// TIA Portal project "KolosCwiczenieSymulatorow" (V14)

(* hardware
DEVICE "S7-1200 station_1"  S7-1200 Station
   slot 0: "Rack_0"  S7-1200 Rack  Rack  V1.0
   slot 1: "PLC_1"  CPU 1214C DC/DC/DC  6ES7 214-1AG40-0XB0  V4.2
DEVICE "HMI_1"  TP700 Comfort
   slot 0: "TP700 Comfort"  TP700 Comfort  6AV2 124-0GC01-0AX0  14.0.1.0
   slot 1: "HMI_RT_1"  TP700 Comfort  6AV2 124-0GC01-0AX0  14.0.1.0
   slot 5: "HMI_1.IE_CP_1"  PROFINET Interface  14.0.1.0
      slot 1: "PROFINET Interface_1"  PROFINET Interface
         slot 1: "Port_1"  Port
         slot 2: "Port_2"  Port
   slot 7: "HMI_1.MPI/DP_CP_1"  MPI/DP Interface  14.0.1.0
*)

// ===== PLC "PLC_1"  CPU 1214C DC/DC/DC =====

VAR_GLOBAL   // PLC tag table "Default tag table"
   "Otworz zawor" AT %Q0.2 : Bool;
   "Zawor Otwarty" AT %I0.1 : Bool;
   "Zawor zamkniety" AT %I0.2 : Bool;
   "Zamknij zawor" AT %Q0.3 : Bool;
   "Dolej" AT %Q0.4 : Bool;
   "Poziom" AT %IW64 : Word;
   "Clock_Byte" AT %MB0 : Byte;
   "Clock_10Hz" AT %M0.0 : Bool;
   "Clock_5Hz" AT %M0.1 : Bool;
   "Clock_2.5Hz" AT %M0.2 : Bool;
   "Clock_2Hz" AT %M0.3 : Bool;
   "Clock_1.25Hz" AT %M0.4 : Bool;
   "Clock_1Hz" AT %M0.5 : Bool;
   "Clock_0.625Hz" AT %M0.6 : Bool;
   "Clock_0.5Hz" AT %M0.7 : Bool;
   "Wypompuj" AT %Q0.5 : Bool;
   "Tag_1" AT %M10.0 : Bool;
   "Tag_2" AT %M10.1 : Bool;
   "Tag_3" AT %IW68 : Word;
   "Tag_4" AT %I10.0 : Bool;
   "Zawor_otwarty" AT %I10.1 : Bool;
   "Zawor_zamkniety" AT %I10.2 : Bool;
   "Tag_5" AT %IW69 : Word;
   "Tag_6" AT %MD30 : DWord;
   "Moc" AT %QW10 : Word;
   "Tag_8" AT %QD10 : Real;
   "Temperatura" AT %ID30 : Real;
   "Tag_10" AT %M10.3 : Bool;
   "Tag_7" AT %IW30 : Word;
   "Tag_9" AT %IW70 : Word;
   "0_krotka" AT %M20.0 : Bool;
   "0_srednia" AT %M20.1 : Bool;
   "0_dluga" AT %M20.2 : Bool;
   "1_krotka" AT %M20.3 : Bool;
   "1_srednia" AT %M20.4 : Bool;
   "1_dluga" AT %M20.5 : Bool;
   "2_krotka" AT %M20.6 : Bool;
   "2_srednia" AT %M20.7 : Bool;
   "2_dluga" AT %M21.0 : Bool;
END_VAR

DATA_BLOCK "Symulator Zaworu_DB"   // DB3
{ S7_Optimized_Access := 'TRUE' }
VERSION : 0.1
// stored: InstanceOfName Symulator Zaworu
"Symulator Zaworu"
BEGIN
END_DATA_BLOCK

DATA_BLOCK "Symulator zaworu 2 cewkowego_DB"   // DB6
{ S7_Optimized_Access := 'TRUE' }
VERSION : 0.1
// stored: InstanceOfName Symulator zaworu 2 cewkowego
"Symulator zaworu 2 cewkowego"
BEGIN
END_DATA_BLOCK

DATA_BLOCK "Symulator Poziomu_DB"   // DB7
{ S7_Optimized_Access := 'TRUE' }
VERSION : 0.1
// stored: InstanceOfName Symulator Poziomu
"Symulator Poziomu"
BEGIN
END_DATA_BLOCK

DATA_BLOCK "Symulator zaworu 2 cewkowego_DB_1"   // DB8
{ S7_Optimized_Access := 'TRUE' }
VERSION : 0.1
// stored: InstanceOfName Symulator zaworu 2 cewkowego
"Symulator zaworu 2 cewkowego"
BEGIN
END_DATA_BLOCK

DATA_BLOCK "Symulator Poziomu_DB_1"   // DB9
{ S7_Optimized_Access := 'TRUE' }
VERSION : 0.1
// stored: InstanceOfName Symulator Poziomu
"Symulator Poziomu"
BEGIN
END_DATA_BLOCK

DATA_BLOCK "Symulator Obiektu Cieplnego_DB"   // DB10
{ S7_Optimized_Access := 'TRUE' }
VERSION : 0.1
// stored: InstanceOfName Symulator Obiektu Cieplnego
"Symulator Obiektu Cieplnego"
BEGIN
END_DATA_BLOCK

// folder: System blocks/Program resources

DATA_BLOCK "IEC_Timer_0_DB"   // DB1
{ S7_Optimized_Access := 'TRUE' }
AUTHOR : Simatic
FAMILY : IEC
NAME : IEC_TMR
VERSION : 1.0
// stored: InstanceOfName IEC_TIMER
"IEC_TIMER"
BEGIN
END_DATA_BLOCK

DATA_BLOCK "IEC_Timer_0_DB_1"   // DB2
{ S7_Optimized_Access := 'TRUE' }
AUTHOR : Simatic
FAMILY : IEC
NAME : IEC_TMR
VERSION : 1.0
// stored: InstanceOfName IEC_TIMER
"IEC_TIMER"
BEGIN
END_DATA_BLOCK

DATA_BLOCK "IEC_Timer_0_DB_2"   // DB4
{ S7_Optimized_Access := 'TRUE' }
AUTHOR : Simatic
FAMILY : IEC
NAME : IEC_TMR
VERSION : 1.0
// stored: InstanceOfName IEC_TIMER
"IEC_TIMER"
BEGIN
END_DATA_BLOCK

DATA_BLOCK "IEC_Timer_0_DB_3"   // DB5
{ S7_Optimized_Access := 'TRUE' }
AUTHOR : Simatic
FAMILY : IEC
NAME : IEC_TMR
VERSION : 1.0
// stored: InstanceOfName IEC_TIMER
"IEC_TIMER"
BEGIN
END_DATA_BLOCK

// folder: (top level)

FUNCTION_BLOCK "Symulator Zaworu"   // FB1, LAD
{ S7_Optimized_Access := 'TRUE' }
VERSION : 0.1
BEGIN

REGION Network 1
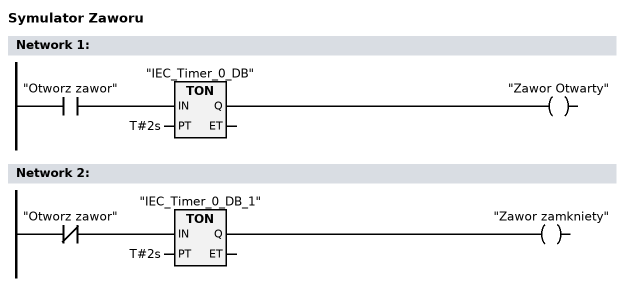
   "IEC_Timer_0_DB".TON(IN := "Otworz zawor", PT := T#2s);
   "Zawor Otwarty" := "IEC_Timer_0_DB".Q;
END_REGION

REGION Network 2
   "IEC_Timer_0_DB_1".TON(IN := NOT "Otworz zawor", PT := T#2s);
   "Zawor zamkniety" := "IEC_Timer_0_DB_1".Q;
END_REGION
END_FUNCTION_BLOCK

FUNCTION_BLOCK "Symulator zaworu 2 cewkowego"   // FB2, LAD
{ S7_Optimized_Access := 'TRUE' }
VERSION : 0.1
   VAR_TEMP   // added for the SCL form of the ladder/FBD networks
      _w1 : Bool;
   END_VAR
BEGIN

REGION Network 1
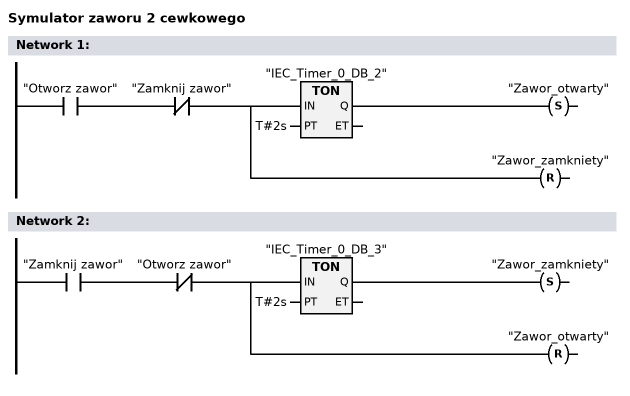
   #_w1 := "Otworz zawor" AND NOT "Zamknij zawor";
   "IEC_Timer_0_DB_2".TON(IN := #_w1, PT := T#2s);
   IF "IEC_Timer_0_DB_2".Q THEN "Zawor_otwarty" := TRUE; END_IF;
   IF #_w1 THEN "Zawor_zamkniety" := FALSE; END_IF;
END_REGION

REGION Network 2
   #_w1 := "Zamknij zawor" AND NOT "Otworz zawor";
   "IEC_Timer_0_DB_3".TON(IN := #_w1, PT := T#2s);
   IF "IEC_Timer_0_DB_3".Q THEN "Zawor_zamkniety" := TRUE; END_IF;
   IF #_w1 THEN "Zawor_otwarty" := FALSE; END_IF;
END_REGION
END_FUNCTION_BLOCK

FUNCTION_BLOCK "Symulator Poziomu"   // FB3, LAD
{ S7_Optimized_Access := 'TRUE' }
VERSION : 0.1
   VAR_TEMP
      Temp_poziom : DInt;
   END_VAR
   VAR CONSTANT
      Delta_dolewania : UInt := 250;
      Delta_wypompowywania : UInt := 500;
   END_VAR
   VAR_TEMP   // added for the SCL form of the ladder/FBD networks
      _w1 : Bool;
   END_VAR
BEGIN

REGION Network 1
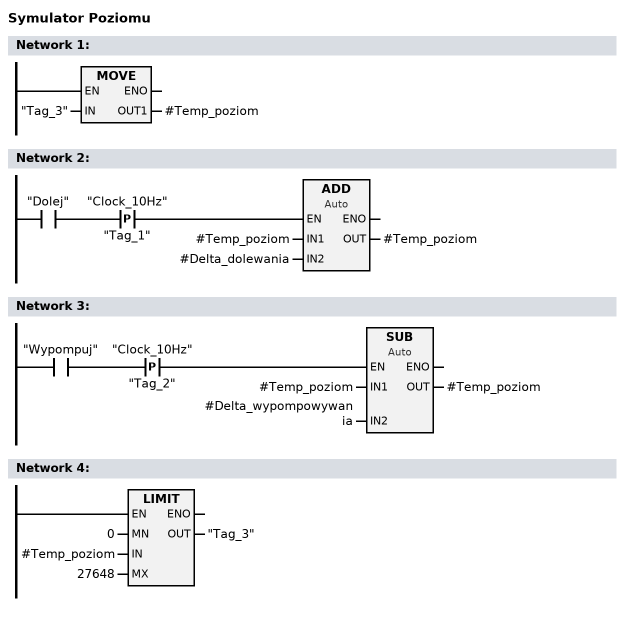
   RUNG wire#powerrail
      Move(in := "Tag_3", out1 => #Temp_poziom)
   END_RUNG
   // the same network as SCL:
   #Temp_poziom := "Tag_3";
END_REGION

REGION Network 2
   RUNG wire#powerrail
      Contact( "Dolej" )
      P_Contact(operand := "Clock_10Hz", bit := "Tag_1")
      Add(in1 := #Temp_poziom, in2 := #Delta_dolewania, out => #Temp_poziom)
   END_RUNG
   // the same network as SCL:
   #_w1 := "Dolej" AND "Clock_10Hz" AND NOT "Tag_1";   // rising edge of "Clock_10Hz"
   "Tag_1" := "Clock_10Hz";
   IF #_w1 THEN #Temp_poziom := #Temp_poziom + #Delta_dolewania; END_IF;
END_REGION

REGION Network 3
   RUNG wire#powerrail
      Contact( "Wypompuj" )
      P_Contact(operand := "Clock_10Hz", bit := "Tag_2")
      Sub(in1 := #Temp_poziom, in2 := #Delta_wypompowywania, out => #Temp_poziom)
   END_RUNG
   // the same network as SCL:
   #_w1 := "Wypompuj" AND "Clock_10Hz" AND NOT "Tag_2";   // rising edge of "Clock_10Hz"
   "Tag_2" := "Clock_10Hz";
   IF #_w1 THEN #Temp_poziom := #Temp_poziom - #Delta_wypompowywania; END_IF;
END_REGION

REGION Network 4
   "Tag_3" := LIMIT(MN := 0, IN := #Temp_poziom, MX := 27648);
END_REGION
END_FUNCTION_BLOCK

FUNCTION_BLOCK "Symulator Obiektu Cieplnego"   // FB4, LAD
{ S7_Optimized_Access := 'TRUE' }
VERSION : 0.1
   VAR_TEMP
      Temp_temperatura : Real;
      Temp_moc : Real;
   END_VAR
   VAR CONSTANT
      Alfa : Real := 0.1;
   END_VAR
   VAR_TEMP   // added for the SCL form of the ladder/FBD networks
      _w1 : Bool;
   END_VAR
BEGIN

REGION Network 1
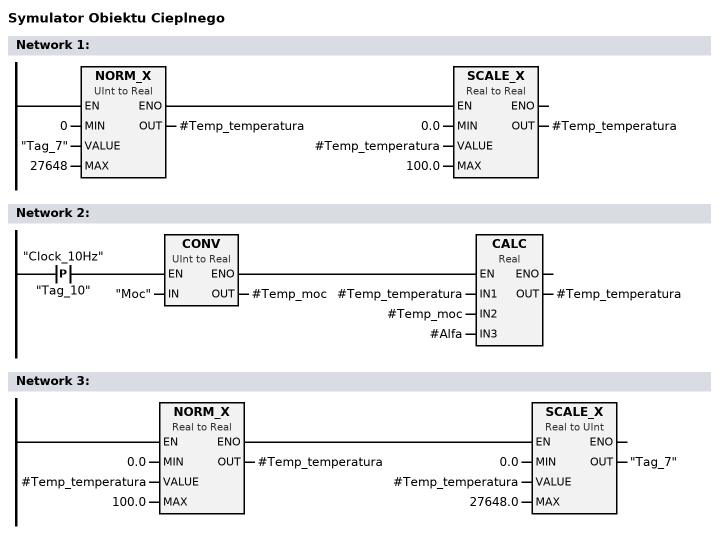
   RUNG wire#powerrail
      { S7_Templates := "[SrcType := UInt, DestType := Real]" } Normalize(min := 0, value := "Tag_7", max := 27648, out => #Temp_temperatura)
      { S7_Templates := "[SrcType := Real, DestType := Real]" } Scale(min := 0.0, value := #Temp_temperatura, max := 100.0, out => #Temp_temperatura)
   END_RUNG
   // the same network as SCL:
   #Temp_temperatura := NORM_X(MIN := 0, VALUE := "Tag_7", MAX := 27648);
   #Temp_temperatura := SCALE_X(MIN := 0.0, VALUE := #Temp_temperatura, MAX := 100.0);
END_REGION

REGION Network 2
   #_w1 := "Clock_10Hz" AND NOT "Tag_10";   // rising edge of "Clock_10Hz"
   "Tag_10" := "Clock_10Hz";
   IF #_w1 THEN
       #Temp_moc := UINT_TO_REAL("Moc");
       CALC(in1 := #Temp_temperatura, in2 := #Temp_moc, in3 := #Alfa, out => #Temp_temperatura);
   END_IF;
END_REGION

REGION Network 3
   RUNG wire#powerrail
      { S7_Templates := "[SrcType := Real, DestType := Real]" } Normalize(min := 0.0, value := #Temp_temperatura, max := 100.0, out => #Temp_temperatura)
      { S7_Templates := "[SrcType := Real, DestType := UInt]" } Scale(min := 0.0, value := #Temp_temperatura, max := 27648.0, out => "Tag_7")
   END_RUNG
   // the same network as SCL:
   #Temp_temperatura := NORM_X(MIN := 0.0, VALUE := #Temp_temperatura, MAX := 100.0);
   "Tag_7" := SCALE_X(MIN := 0.0, VALUE := #Temp_temperatura, MAX := 27648.0);
END_REGION
END_FUNCTION_BLOCK

ORGANIZATION_BLOCK "Main"   // OB1, LAD, ProgramCycle
TITLE = "Main Program Sweep (Cycle)"
{ S7_Optimized_Access := 'TRUE' }
VERSION : 0.1
   VAR_INPUT
      Initial_Call : Bool;   // Initial call of this OB
      Remanence : Bool;   // =True, if remanent data are available
   END_VAR
BEGIN
END_ORGANIZATION_BLOCK

(* ===== HMI "HMI_RT_1" =====
system functions are stored by id; their names below are inferred from use
connection "HMI_Connection_1": ETHERNET, S7_1200_OMS

HMI tags "Default tag table"
   "Tag_ScreenNumber" : UInt, internal
   "0_krotka" : Bool = PLC 0_krotka AT %M20.0, 100 ms
   "0_srednia" : Bool = PLC 0_srednia AT %M20.1, 100 ms
   "0_dluga" : Bool = PLC 0_dluga AT %M20.2, 100 ms
   "1_krotka" : Bool = PLC 1_krotka AT %M20.3, 100 ms
   "1_srednia" : Bool = PLC 1_srednia AT %M20.4, 100 ms
   "1_dluga" : Bool = PLC 1_dluga AT %M20.5, 100 ms
   "2_krotka" : Bool = PLC 2_krotka AT %M20.6, 100 ms
   "2_srednia" : Bool = PLC 2_srednia AT %M20.7, 100 ms
   "2_dluga" : Bool = PLC 2_dluga AT %M21.0, 100 ms

Template "Template_1" 800x480
   Button "Exit" at 714,429 size 71x50; TextOff 'Exit'; PictureOff "ExitRuntime_KTP700_Basic_DP_TR"; PictureOn "ExitRuntime_KTP700_Basic_DP_TR"
      on Release: StopRuntime(0)
   Button "Template_Button" at 614,429 size 71x50; TextOff 'Text'
   Button "Template_Button_1" at 514,429 size 71x50; TextOff 'Text'
   Button "Template_Button_2" at 414,429 size 71x50; TextOff 'Text'
   Button "Template_Button_3" at 314,429 size 71x50; TextOff 'Text'
   Button "Template_Button_4" at 214,429 size 71x50; TextOff 'Text'
   Button "Template_Button_5" at 114,429 size 71x50; TextOff 'Text'
   Button "Start screen" at 14,429 size 71x50; TextOff 'Start screen'; PictureOff "NavigateHome_KTP700_Basic_DP_TR"; PictureOn "NavigateHome_KTP700_Basic_DP_TR"
      on Release: ActivateScreen("Root screen", 0)
   SymbolicIOField "Symbolic_IO_Field_Screen" at 93,9 size 600x33; TextOff '0'; TextOn '1'; TextList "TextList_ScreenNames"
      ProcessValue <- "Tag_ScreenNumber"
      on Change: ActivateScreenByNumber("Tag_ScreenNumber", 0)
   DateTimeField "HmiScreenItemData" at 695,25 size 105x25
   DateTimeField "HmiScreenItemData_1" at 695,0 size 105x25
   GraphicView "Logo" at 0,0 size 91x51; Picture "Logo of HMI_1"

screen "Root screen" 800x480, template "Template_1"
   on GenerateScreen: SetTag("Tag_ScreenNumber", 1)
   Switch "l_kr" at 365,86 size 50x50; CaptionText 'Switch'; TextOff '0'; TextOn '1'; PictureOff "Pushbutton_Round_G_Off_256c"; PictureOn "Pushbutton_Round_G_On_256c"
      ProcessValue <- "0_krotka"
      on SwitchOn: "Przypisanie_belki_do_zsypu"('krotka', 'lewy')
      on SwitchOff: "Odpiecie_belki_do_zsypu"('krotka', 'lewy')
   Switch "l_sr" at 365,137 size 50x50; CaptionText 'Switch'; TextOff '0'; TextOn '1'; PictureOff "Pushbutton_Round_GN_Off_256c"; PictureOn "Pushbutton_Round_GN_On_256c"
      ProcessValue <- "0_srednia"
      on SwitchOn: "Przypisanie_belki_do_zsypu"('srednia', 'lewy')
      on SwitchOff: "Odpiecie_belki_do_zsypu"('srednia', 'lewy')
   Switch "l_dl" at 365,188 size 50x50; CaptionText 'Switch'; TextOff '0'; TextOn '1'; PictureOff "Pushbutton_Round_R_Off_256c"; PictureOn "Pushbutton_Round_R_On_256c"
      ProcessValue <- "0_dluga"
      on SwitchOn: "Przypisanie_belki_do_zsypu"('dluga', 'lewy')
      on SwitchOff: "Odpiecie_belki_do_zsypu"('dluga', 'lewy')
   Switch "s_kr" at 473,87 size 50x50; CaptionText 'Switch'; TextOff '0'; TextOn '1'; PictureOff "Pushbutton_Round_G_Off_256c"; PictureOn "Pushbutton_Round_G_On_256c"
      ProcessValue <- "1_krotka"
      on SwitchOn: "Przypisanie_belki_do_zsypu"('krotka', 'srodkowy')
      on SwitchOff: "Odpiecie_belki_do_zsypu"('krotka', 'srodkowy')
   Switch "s_sr" at 473,138 size 50x50; CaptionText 'Switch'; TextOff '0'; TextOn '1'; PictureOff "Pushbutton_Round_GN_Off_256c"; PictureOn "Pushbutton_Round_GN_On_256c"
      ProcessValue <- "1_srednia"
      on SwitchOn: "Przypisanie_belki_do_zsypu"('srednia', 'srodkowy')
      on SwitchOff: "Odpiecie_belki_do_zsypu"('srednia', 'srodkowy')
   Switch "s_dl" at 473,189 size 50x50; CaptionText 'Switch'; TextOff '0'; TextOn '1'; PictureOff "Pushbutton_Round_R_Off_256c"; PictureOn "Pushbutton_Round_R_On_256c"
      ProcessValue <- "1_dluga"
      on SwitchOn: "Przypisanie_belki_do_zsypu"('dluga', 'srodkowy')
      on SwitchOff: "Odpiecie_belki_do_zsypu"('dluga', 'srodkowy')
   Switch "p_kr" at 573,89 size 50x50; CaptionText 'Switch'; TextOff '0'; TextOn '1'; PictureOff "Pushbutton_Round_G_Off_256c"; PictureOn "Pushbutton_Round_G_On_256c"
      on SwitchOn: "Przypisanie_belki_do_zsypu"('krotka', 'prawy')
      ProcessValue <- "2_krotka"
      on SwitchOff: "Odpiecie_belki_do_zsypu"('krotka', 'prawy')
   Switch "p_sr" at 573,140 size 50x50; CaptionText 'Switch'; TextOff '0'; TextOn '1'; PictureOff "Pushbutton_Round_GN_Off_256c"; PictureOn "Pushbutton_Round_GN_On_256c"
      on SwitchOn: "Przypisanie_belki_do_zsypu"('srednia', 'prawy')
      ProcessValue <- "2_srednia"
      on SwitchOff: "Odpiecie_belki_do_zsypu"('srednia', 'prawy')
   Switch "p_dl" at 573,191 size 50x50; CaptionText 'Switch'; TextOff '0'; TextOn '1'; PictureOff "Pushbutton_Round_R_Off_256c"; PictureOn "Pushbutton_Round_R_On_256c"
      on SwitchOn: "Przypisanie_belki_do_zsypu"('dluga', 'prawy')
      ProcessValue <- "2_dluga"
      on SwitchOff: "Odpiecie_belki_do_zsypu"('dluga', 'prawy')
   TextField "text_lewy" at 361,238 size 67x67; Text 'Text'
   TextField "text_srodkowy" at 458,243 size 73x59; Text 'Text'
   TextField "text_prawy" at 564,239 size 65x75; Text 'Text'

VB script "Przypisanie_belki_do_zsypu"
   'Zsyp: 				0			1			2
   'Rozmiar belki:		0_krotka	1_krotka	2_krotka
   '					0_srednia	1_srednia	2_srednia
   '					0_dluga		1_dluga		2_dluga
   
   If zsyp = "lewy" Then
   	If dlugosc_belki = "krotka" Then	'jezeli wybrano rozmiar belki krotki
   		HmiRuntime.Screens("Root screen").ScreenItems("text_lewy").Text = "pnie" & Chr(10) & "krótkie"	'ustaw na zsypie informacje o wybranej belce 
   		HmiRuntime.Screens("Root screen").ScreenItems("l_sr").Enabled = False
   		HmiRuntime.Screens("Root screen").ScreenItems("l_dl").Enabled = False							
   		HmiRuntime.Screens("Root screen").ScreenItems("s_kr").Enabled = False							
   		HmiRuntime.Screens("Root screen").ScreenItems("p_kr").Enabled = False
   	ElseIf dlugosc_belki = "srednia" Then
   		HmiRuntime.Screens("Root screen").ScreenItems("text_lewy").Text = "pnie" & Chr(10) & "średnie" 
   		HmiRuntime.Screens("Root screen").ScreenItems("l_kr").Enabled = False
   		HmiRuntime.Screens("Root screen").ScreenItems("l_dl").Enabled = False
   		HmiRuntime.Screens("Root screen").ScreenItems("s_sr").Enabled = False
   		HmiRuntime.Screens("Root screen").ScreenItems("p_sr").Enabled = False
   	ElseIf dlugosc_belki = "dluga" Then
   		HmiRuntime.Screens("Root screen").ScreenItems("text_lewy").Text = "pnie" & Chr(10) & "długie" 
   		HmiRuntime.Screens("Root screen").ScreenItems("l_kr").Enabled = False
   		HmiRuntime.Screens("Root screen").ScreenItems("l_sr").Enabled = False
   		HmiRuntime.Screens("Root screen").ScreenItems("s_dl").Enabled = False
   		HmiRuntime.Screens("Root screen").ScreenItems("p_dl").Enabled = False
   	End If
   ElseIf zsyp = "srodkowy" Then
   	If dlugosc_belki = "krotka" Then
   		HmiRuntime.Screens("Root screen").ScreenItems("text_srodkowy").Text = "pnie" & Chr(10) & "krótkie" 
   		HmiRuntime.Screens("Root screen").ScreenItems("s_sr").Enabled = False
   		HmiRuntime.Screens("Root screen").ScreenItems("s_dl").Enabled = False
   		HmiRuntime.Screens("Root screen").ScreenItems("l_kr").Enabled = False
   		HmiRuntime.Screens("Root screen").ScreenItems("p_kr").Enabled = False
   	ElseIf dlugosc_belki = "srednia" Then
   		HmiRuntime.Screens("Root screen").ScreenItems("text_srodkowy").Text = "pnie" & Chr(10) & "średnie" 
   		HmiRuntime.Screens("Root screen").ScreenItems("s_kr").Enabled = False
   		HmiRuntime.Screens("Root screen").ScreenItems("s_dl").Enabled = False
   		HmiRuntime.Screens("Root screen").ScreenItems("l_sr").Enabled = False
   		HmiRuntime.Screens("Root screen").ScreenItems("p_sr").Enabled = False
   	ElseIf dlugosc_belki = "dluga" Then
   		HmiRuntime.Screens("Root screen").ScreenItems("text_srodkowy").Text = "pnie" & Chr(10) & "długie" 
   		HmiRuntime.Screens("Root screen").ScreenItems("s_kr").Enabled = False
   		HmiRuntime.Screens("Root screen").ScreenItems("s_sr").Enabled = False
   		HmiRuntime.Screens("Root screen").ScreenItems("l_dl").Enabled = False
   		HmiRuntime.Screens("Root screen").ScreenItems("p_dl").Enabled = False
   	End If
   ElseIf zsyp = "prawy" Then
   	If dlugosc_belki = "krotka" Then
   		HmiRuntime.Screens("Root screen").ScreenItems("text_prawy").Text = "pnie" & Chr(10) & "krótkie" 
   		HmiRuntime.Screens("Root screen").ScreenItems("p_sr").Enabled = False
   		HmiRuntime.Screens("Root screen").ScreenItems("p_dl").Enabled = False
   		HmiRuntime.Screens("Root screen").ScreenItems("l_kr").Enabled = False
   		HmiRuntime.Screens("Root screen").ScreenItems("s_kr").Enabled = False
   	ElseIf dlugosc_belki = "srednia" Then
   		HmiRuntime.Screens("Root screen").ScreenItems("text_prawy").Text = "pnie" & Chr(10) & "średnie" 
   		HmiRuntime.Screens("Root screen").ScreenItems("p_kr").Enabled = False
   		HmiRuntime.Screens("Root screen").ScreenItems("p_dl").Enabled = False
   		HmiRuntime.Screens("Root screen").ScreenItems("l_sr").Enabled = False
   		HmiRuntime.Screens("Root screen").ScreenItems("s_sr").Enabled = False
   	ElseIf dlugosc_belki = "dluga" Then
   		HmiRuntime.Screens("Root screen").ScreenItems("text_prawy").Text = "pnie" & Chr(10) & "długie" 
   		HmiRuntime.Screens("Root screen").ScreenItems("p_kr").Enabled = False
   		HmiRuntime.Screens("Root screen").ScreenItems("p_sr").Enabled = False
   		HmiRuntime.Screens("Root screen").ScreenItems("l_dl").Enabled = False
   		HmiRuntime.Screens("Root screen").ScreenItems("s_dl").Enabled = False
   	End If
   End If

VB script "Odpiecie_belki_do_zsypu"
   If zsyp = "lewy" Then
   	If dlugosc_belki = "krotka" Then	'jezeli wybrano rozmiar belki krotki
   		HmiRuntime.Screens("Root screen").ScreenItems("text_lewy").Text = "pnie" & Chr(10) & "-----" 
   		If Not SmartTags("1_srednia") And Not SmartTags("2_srednia") Then
   			HmiRuntime.Screens("Root screen").ScreenItems("l_sr").Enabled = True							
   		End If
   		If Not SmartTags("1_dluga") And Not SmartTags("2_dluga") Then
   			HmiRuntime.Screens("Root screen").ScreenItems("l_dl").Enabled = True
   		End If
   		If Not SmartTags("1_srednia") And Not SmartTags("1_dluga") Then							
   			HmiRuntime.Screens("Root screen").ScreenItems("s_kr").Enabled = True
   		End If
   		If Not SmartTags("2_srednia") And Not SmartTags("2_dluga") Then
   			HmiRuntime.Screens("Root screen").ScreenItems("p_kr").Enabled = True
   		End If							
   	ElseIf dlugosc_belki = "srednia" Then
   		HmiRuntime.Screens("Root screen").ScreenItems("text_lewy").Text = "pnie" & Chr(10) & "-----"
   		If Not SmartTags("1_krotka") And Not SmartTags("2_krotka") Then
   			HmiRuntime.Screens("Root screen").ScreenItems("l_kr").Enabled = True
   		End If
   		If Not SmartTags("1_dluga") And Not SmartTags("2_dluga") Then
   			HmiRuntime.Screens("Root screen").ScreenItems("l_dl").Enabled = True
   		End If
   		If Not SmartTags("1_krotka") And Not SmartTags("1_dluga") Then
   			HmiRuntime.Screens("Root screen").ScreenItems("s_sr").Enabled = True
   		End If
   		If Not SmartTags("2_krotka") And Not SmartTags("2_dluga") Then
   			HmiRuntime.Screens("Root screen").ScreenItems("p_sr").Enabled = True
   		End If
   	ElseIf dlugosc_belki = "dluga" Then
   		HmiRuntime.Screens("Root screen").ScreenItems("text_lewy").Text = "pnie" & Chr(10) & "-----" 
   		If Not SmartTags("1_krotka") And Not SmartTags("2_krotka") Then
   			HmiRuntime.Screens("Root screen").ScreenItems("l_kr").Enabled = True
   		End If
   		If Not SmartTags("1_srednia") And Not SmartTags("2_srednia") Then
   			HmiRuntime.Screens("Root screen").ScreenItems("l_sr").Enabled = True
   		End If
   		If Not SmartTags("1_krotka") And Not SmartTags("1_srednia") Then
   			HmiRuntime.Screens("Root screen").ScreenItems("s_dl").Enabled = True
   		End If
   		If Not SmartTags("2_krotka") And Not SmartTags("2_srednia") Then
   			HmiRuntime.Screens("Root screen").ScreenItems("p_dl").Enabled = True
   		End If
   	End If
   ElseIf zsyp = "srodkowy" Then
   	If dlugosc_belki = "krotka" Then
   		HmiRuntime.Screens("Root screen").ScreenItems("text_srodkowy").Text = "pnie" & Chr(10) & "-----"
   		If Not SmartTags("0_srednia") And Not SmartTags("2_srednia") Then
   			HmiRuntime.Screens("Root screen").ScreenItems("s_sr").Enabled = True
   		End If
   		If Not SmartTags("0_dluga") And Not SmartTags("2_dluga") Then
   			HmiRuntime.Screens("Root screen").ScreenItems("s_dl").Enabled = True
   		End If
   		If Not SmartTags("0_srednia") And Not SmartTags("0_dluga") Then
   			HmiRuntime.Screens("Root screen").ScreenItems("l_kr").Enabled = True
   		End If
   		If Not SmartTags("2_srednia") And Not SmartTags("2_dluga") Then
   			HmiRuntime.Screens("Root screen").ScreenItems("p_kr").Enabled = True
   		End If
   	ElseIf dlugosc_belki = "srednia" Then
   		HmiRuntime.Screens("Root screen").ScreenItems("text_srodkowy").Text = "pnie" & Chr(10) & "-----" 
   		If Not SmartTags("0_krotka") And Not SmartTags("2_krotka") Then
   			HmiRuntime.Screens("Root screen").ScreenItems("s_kr").Enabled = True
   		End If
   		If Not SmartTags("0_dluga") And Not SmartTags("2_dluga") Then
   			HmiRuntime.Screens("Root screen").ScreenItems("s_dl").Enabled = True
   		End If
   		If Not SmartTags("0_krotka") And Not SmartTags("1_dluga") Then
   			HmiRuntime.Screens("Root screen").ScreenItems("l_sr").Enabled = True
   		End If
   		If Not SmartTags("2_krotka") And Not SmartTags("2_dluga") Then
   			HmiRuntime.Screens("Root screen").ScreenItems("p_sr").Enabled = True
   		End If
   	ElseIf dlugosc_belki = "dluga" Then
   		HmiRuntime.Screens("Root screen").ScreenItems("text_srodkowy").Text = "pnie" & Chr(10) & "-----"
   		If Not SmartTags("0_krotka") And Not SmartTags("2_krotka") Then
   			HmiRuntime.Screens("Root screen").ScreenItems("s_kr").Enabled = True
   		End If
   		If Not SmartTags("0_srednia") And Not SmartTags("2_srednia") Then
   			HmiRuntime.Screens("Root screen").ScreenItems("s_sr").Enabled = True
   		End If
   		If Not SmartTags("0_krotka") And Not SmartTags("0_srednia") Then
   			HmiRuntime.Screens("Root screen").ScreenItems("l_dl").Enabled = True
   		End If
   		If Not SmartTags("2_krotka") And Not SmartTags("2_srednia") Then
   			HmiRuntime.Screens("Root screen").ScreenItems("p_dl").Enabled = True
   		End If
   	End If
   ElseIf zsyp = "prawy" Then
   	If dlugosc_belki = "krotka" Then
   		HmiRuntime.Screens("Root screen").ScreenItems("text_prawy").Text = "pnie" & Chr(10) & "-----"
   		If Not SmartTags("0_srednia") And Not SmartTags("1_srednia") Then
   			HmiRuntime.Screens("Root screen").ScreenItems("p_sr").Enabled = True
   		End If
   		If Not SmartTags("0_dluga") And Not SmartTags("1_dluga") Then
   			HmiRuntime.Screens("Root screen").ScreenItems("p_dl").Enabled = True
   		End If
   		If Not SmartTags("0_srednia") And Not SmartTags("0_dluga") Then
   			HmiRuntime.Screens("Root screen").ScreenItems("l_kr").Enabled = True
   		End If
   		If Not SmartTags("1_srednia") And Not SmartTags("1_dluga") Then
   			HmiRuntime.Screens("Root screen").ScreenItems("s_kr").Enabled = True
   		End If
   	ElseIf dlugosc_belki = "srednia" Then
   		HmiRuntime.Screens("Root screen").ScreenItems("text_prawy").Text = "pnie" & Chr(10) & "-----" 
   		If Not SmartTags("0_krotka") And Not SmartTags("1_krotka") Then
   			HmiRuntime.Screens("Root screen").ScreenItems("p_kr").Enabled = True
   		End If
   		If Not SmartTags("0_dluga") And Not SmartTags("1_dluga") Then
   			HmiRuntime.Screens("Root screen").ScreenItems("p_dl").Enabled = True
   		End If
   		If Not SmartTags("0_krotka") And Not SmartTags("0_dluga") Then
   			HmiRuntime.Screens("Root screen").ScreenItems("l_sr").Enabled = True
   		End If
   		If Not SmartTags("1_krotka") And Not SmartTags("1_dluga") Then
   			HmiRuntime.Screens("Root screen").ScreenItems("s_sr").Enabled = True
   		End If
   	ElseIf dlugosc_belki = "dluga" Then
   		HmiRuntime.Screens("Root screen").ScreenItems("text_prawy").Text = "pnie" & Chr(10) & "-----"
   		If Not SmartTags("0_krotka") And Not SmartTags("1_krotka") Then
   			HmiRuntime.Screens("Root screen").ScreenItems("p_kr").Enabled = True
   		End If
   		If Not SmartTags("0_srednia") And Not SmartTags("1_srednia") Then
   			HmiRuntime.Screens("Root screen").ScreenItems("p_sr").Enabled = True
   		End If
   		If Not SmartTags("0_krotka") And Not SmartTags("0_srednia") Then
   			HmiRuntime.Screens("Root screen").ScreenItems("l_dl").Enabled = True
   		End If
   		If Not SmartTags("1_krotka") And Not SmartTags("1_srednia") Then
   			HmiRuntime.Screens("Root screen").ScreenItems("s_dl").Enabled = True
   		End If 	
   	End If
   End If
*)